// TIA Portal V18 export
FUNCTION "IAI" : Void   // FC2200, LAD
{ S7_Optimized_Access := 'TRUE' }
VERSION : 0.1
// stored: AutoNumber false, IsIECCheckEnabled false, SetENOAutomatically false, UDAEnableTagReadback false
BEGIN

REGION Network 1 (SCL): 模式 / Mode
   "ModeDB".Gen.Out.Estop := "Station_Sys".Status.EStopOK;
   "ModeDB".Gen.Out.Reset := "Station_Sys".Cmd.Reset;
   "ModeDB".Gen.Out.Manual := "Station_Sys".Manual.Mode;
   "ModeDB".Gen.Out.Auto := "Station_Sys".Auto.Mode;
   "ModeDB".Gen.Out.Home := "Station_Sys".Initial.Running;
   "ModeDB".Gen.Out.Running := "Station_Sys".Auto.Mode;//"Station_Sys".Auto.Running OR "ST10_PM".Num[7].InitialRun;
   //"ModeDB".Gen.Out.Change:=
END_REGION

REGION Network 2
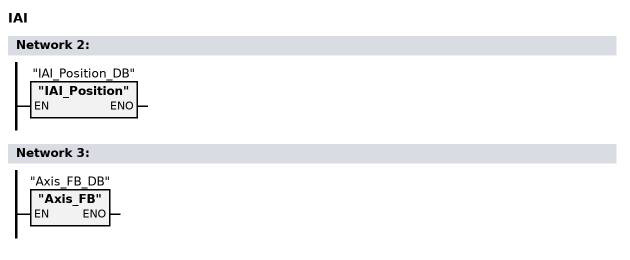
   RUNG wire#powerrail
      "IAI_Position_DB"()
   END_RUNG
   // the same network as SCL:
   "IAI_Position_DB"();   // "IAI_Position"
END_REGION

REGION Network 3
   RUNG wire#powerrail
      "Axis_FB_DB"()
   END_RUNG
   // the same network as SCL:
   "Axis_FB_DB"();   // "Axis_FB"
END_REGION
END_FUNCTION
